FUNCTION_BLOCK Byte2Double (* Basic Function Block Type *)
  (* Standard: 61499-2 *)
  (* Version 0.0, 12/6/2015, gulzha, nxtControl GmbH, Template *)
  PACKAGE Main;
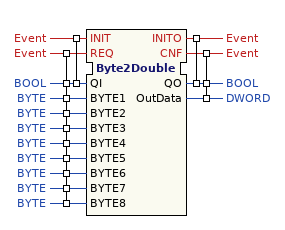
  EVENT_INPUT
    INIT WITH QI; (* Initialization Request *)
    REQ WITH QI, BYTE1, BYTE2, BYTE3, BYTE4, BYTE5, BYTE6, BYTE7, BYTE8; (* Normal Execution Request *)
  END_EVENT
  EVENT_OUTPUT
    INITO WITH QO; (* Initialization Confirm *)
    CNF WITH QO, OutData; (* Execution Confirmation *)
  END_EVENT
  VAR_INPUT
    QI : BOOL; (* Input event qualifier *)
    BYTE1 : BYTE;
    BYTE2 : BYTE;
    BYTE3 : BYTE;
    BYTE4 : BYTE;
    BYTE5 : BYTE;
    BYTE6 : BYTE;
    BYTE7 : BYTE;
    BYTE8 : BYTE;
  END_VAR
  VAR_OUTPUT
    QO : BOOL; (* Output event qualifier *)
    OutData : DWORD;
  END_VAR
  VAR
    temp : DWORD;
    i : INT;
    tempByte : BYTE;
  END_VAR
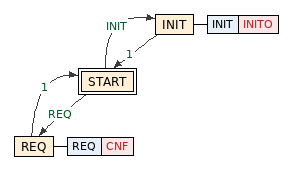
  EC_STATES
    START; (* Initial State *)
    INIT : INIT -> INITO; (* Initialization *)
    REQ : REQ -> CNF; (* Normal execution *)
  END_STATES
  EC_TRANSITIONS
    START TO INIT := INIT;
    INIT TO START := 1;
    START TO REQ := REQ;
    REQ TO START := 1;
  END_TRANSITIONS
  ALGORITHM INIT IN ST: (* Initialization algorithm *)
;
  END_ALGORITHM
  ALGORITHM REQ IN ST: (* Normally executed algorithm *)
;

temp := 0;
//4bytesData := (SHL(SHL(SHL(BYTE_TO_DWORD(in1), 8) OR BYTE_TO_DWORD(in2), 8) OR     BYTE_TO_DWORD(in3), 8) OR in4);

//temp:= BYTE_TO_LREAL(Inputarray[0])
temp:= ((*SHL((temp OR BYTE_TO_LREAL(BYTE1)),56) OR SHL((temp OR BYTE_TO_LREAL(BYTE2)),48) OR
        SHL((temp OR BYTE_TO_LREAL(BYTE3)),40) OR SHL((temp OR BYTE_TO_LREAL(BYTE4)),32) OR*)
        SHL((temp OR BYTE_TO_DWORD(BYTE5)),24) OR SHL((temp OR BYTE_TO_DWORD(BYTE6)),16) OR
        SHL((temp OR BYTE_TO_DWORD(BYTE7)),8) OR (temp OR BYTE_TO_DWORD(BYTE1)));
OutData:=temp;
//OutData:= ; //LREAL_TO_DWORD();
  END_ALGORITHM
END_FUNCTION_BLOCK
